FUNCTION_BLOCK RotatingArmControl (* Basic Function Block Type *)
  (* Standard: 61499-2 *)
  (* Version 0.0, 2/9/2018, Sandeep Patil, nxtControl GmbH, Template *)
  PACKAGE Main;
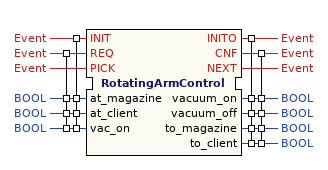
  EVENT_INPUT
    INIT WITH at_magazine, at_client, vac_on; (* Initialization Request *)
    REQ WITH at_magazine, at_client, vac_on; (* Normal Execution Request *)
    PICK;
  END_EVENT
  EVENT_OUTPUT
    INITO WITH vacuum_on, vacuum_off, to_magazine, to_client; (* Initialization Confirm *)
    CNF WITH vacuum_on, vacuum_off, to_magazine, to_client; (* Execution Confirmation *)
    NEXT;
  END_EVENT
  VAR_INPUT
    at_magazine : BOOL; (* Input event qualifier *)
    at_client : BOOL;
    vac_on : BOOL;
  END_VAR
  VAR_OUTPUT
    vacuum_on : BOOL; (* Output event qualifier *)
    vacuum_off : BOOL;
    to_magazine : BOOL;
    to_client : BOOL;
  END_VAR
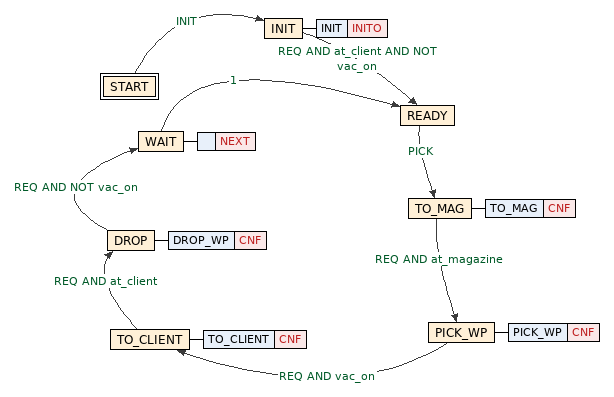
  EC_STATES
    START; (* Initial State *)
    INIT : INIT -> INITO; (* Initialization *)
    DROP : DROP_WP -> CNF; (* Normal execution *)
    READY;
    TO_MAG : TO_MAG -> CNF;
    PICK_WP : PICK_WP -> CNF;
    TO_CLIENT : TO_CLIENT -> CNF;
    WAIT : -> NEXT;
  END_STATES
  EC_TRANSITIONS
    START TO INIT := INIT;
    INIT TO READY := REQ AND at_client AND NOT vac_on;
    READY TO TO_MAG := PICK;
    TO_MAG TO PICK_WP := REQ AND at_magazine;
    PICK_WP TO TO_CLIENT := REQ AND vac_on;
    TO_CLIENT TO DROP := REQ AND at_client;
    DROP TO WAIT := REQ AND NOT vac_on;
    WAIT TO READY := 1;
  END_TRANSITIONS
  ALGORITHM INIT IN ST: (* Initialization algorithm *)
to_client := TRUE;
vacuum_off := TRUE;
vacuum_on := FALSE;
to_magazine := FALSE;
  END_ALGORITHM
  ALGORITHM PICK_WP IN ST: (* Normally executed algorithm *)
vacuum_on := TRUE;
to_magazine := FALSE;
  END_ALGORITHM
  ALGORITHM TO_MAG IN ST:
to_magazine := TRUE;
to_client := FALSE;
vacuum_off := FALSE;
  END_ALGORITHM
  ALGORITHM TO_CLIENT IN ST:
to_magazine := FALSE;
to_client := TRUE;
  END_ALGORITHM
  ALGORITHM DROP_WP IN ST:
vacuum_off := TRUE;
  END_ALGORITHM
END_FUNCTION_BLOCK
